FUNCTION Convert_LWORD_TO_USINT : Hresult
VAR_INPUT
	in : LWORD;
	out : REFERENCE TO USINT;
END_VAR
VAR
	converted : USINT;
END_VAR
VAR CONSTANT
	INCOMPATIBLE : HRESULT := 16#9811070E;
END_VAR

converted := LWORD_TO_USINT(in);

IF (USINT_TO_LWORD(converted) <> in) THEN
	Convert_LWORD_TO_USINT := INCOMPATIBLE;
	RETURN;
END_IF

out := converted;

END_FUNCTION

(* stored: Version 1.1.0.1, ProductVersion 3.1.4024.12
   POU Convert_LWORD_TO_USINT: Id {28a5d013-ad45-4318-bb83-dd25fbc0773c}, SpecialFunc None *)
